(* PLC project Generated.project, CODESYS CODESYS V3.5 SP19 Patch 1 *)
(* stored: creationDateTime 2026-08-18T01:35:02.832885, modificationDateTime 2026-08-18T01:35:02.832885 *)

(* ═══════════════════════════════════════════════════════════════ ST_WinchCfg — Configurations et paramètres réglables pour un Treuil M1/M2 ─────────────────────────────────────────────────────────────── 🎨 Destiné au paramétrage et calibration depuis l'IHM (RETAIN). ═══════════════════════════════════════════════════════════════ *)
TYPE ST_WinchCfg : STRUCT
  CfgTopSensorPos_M : REAL := 8.5;  (* 📐 Position cible du capteur haut (m) *)
  CfgHomingTarget_M : REAL := 0;  (* Cible libre Homing unitaire MAINT_N2 [-99..+99 m] *)
  CfgRampAccelRate : REAL := 50;  (* 📈 Rampe d'accélération (%/s) *)
  CfgRampDecelNormalRate : REAL := 150;  (* 📉 Rampe de décélération normale (%/s) *)
  CfgRampDecelFastRate : REAL := 400;  (* ⚡ Rampe de décélération rapide / SafeStop (%/s) *)
  CfgCableLimitDescent_M : REAL := -20;  (* 📐 Limite basse physique de descente (m, négatif) *)
  Initialized : BOOL := FALSE;  (* 🚦 Flag restauration boot — défaut FALSE non ambigu 🚦 TRUE = config restaurée depuis GVL_PERSISTENT ce boot *)
END_STRUCT;
END_TYPE

(* ======================================================================= 💾 FB_CfgPersistBridge_WinchCfg — Pont persistance pour ST_WinchCfg ─────────────────────────────────────────────────────────────── 🎯 Rôle : Restauration et synchronisation bidirectionnelle IHM / Persist 💾 Persistance : Transfert GVL_PERSISTENT <-> GVL_IHM sur Initialized 📄 Doc métier : DOC/AF/AF_Partie-10_Fonction_Winch_v2.0.md ======================================================================= *)
FUNCTION_BLOCK FB_CfgPersistBridge_WinchCfg
  VAR_OUTPUT
    JustRestored : BOOL;  (* === ETATS RESTAURATION === <-- [STAT] Vrai sur le cycle de restauration initiale *)
  END_VAR
  VAR_IN_OUT
    Hmi : ST_WinchCfg;  (* === BUS CONFIGURATION ET PERSISTANCE === <-> [BUS] Structure de configuration IHM *)
    Persist : ST_WinchCfg;  (* <-> [BUS] Structure de configuration persistante *)
  END_VAR

            

JustRestored := FALSE;
IF NOT Hmi.Initialized THEN
    Hmi := Persist;
    Hmi.Initialized := TRUE;
    JustRestored := TRUE;
ELSE
    Persist := Hmi;
END_IF;

          
END_FUNCTION_BLOCK
